// TIA Portal V18 export
FUNCTION_BLOCK "LEDS"   // FB17, LAD
{ S7_Optimized_Access := 'TRUE' }
// stored: AutoNumber false, MemoryReserve 100, SetENOAutomatically false
   VAR
      ElevClLEDStatus : Bool;
      MSVClLEDStatus : Bool;
      BUWClLEDStatus : Bool;
   END_VAR
   VAR_TEMP
      BUWClLEDOffDely : Bool;
   END_VAR
BEGIN

REGION Network 1: Elev Closed LED
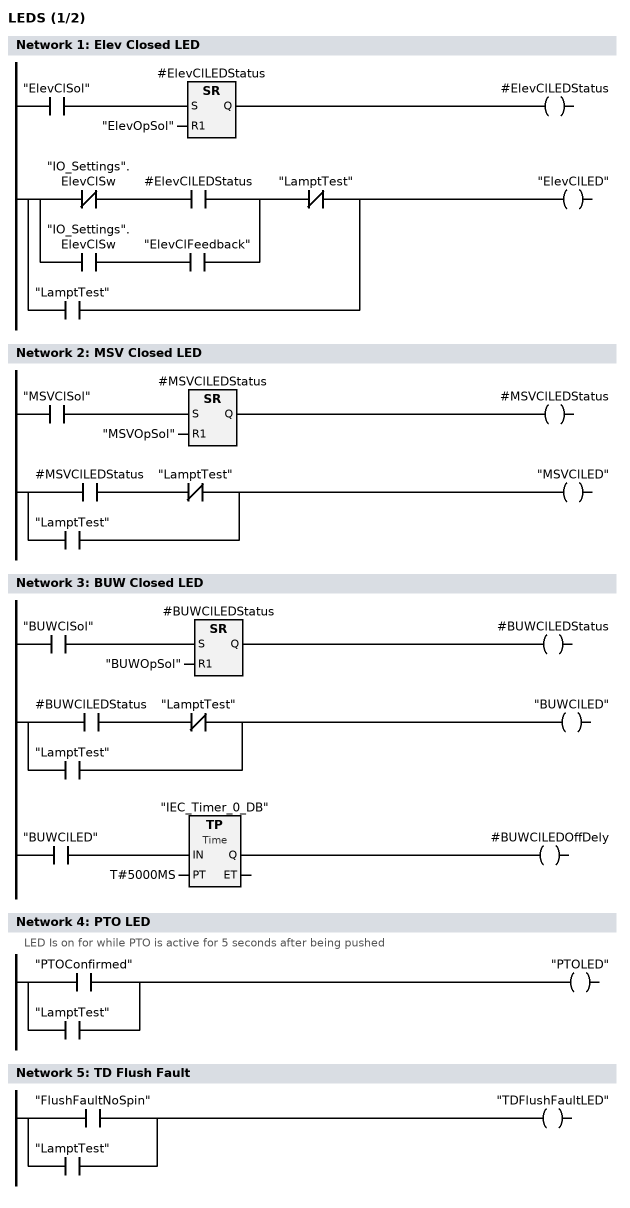
   RUNG wire#powerrail
      Contact( "ElevClSol" )
      S_SR(operand := #ElevClLEDStatus, r1 := "ElevOpSol")
      Coil( #ElevClLEDStatus )
   END_RUNG
   RUNG wire#powerrail
      I_Contact( "IO_Settings".ElevClSw )
      Contact( #ElevClLEDStatus )
      wire#w1
      I_Contact( "LamptTest" )
      wire#w2
      Coil( "ElevClLED" )
   END_RUNG
   RUNG wire#powerrail
      Contact( "IO_Settings".ElevClSw )
      Contact( "ElevClFeedback" )
   END_RUNG wire#w1
   RUNG wire#powerrail
      Contact( "LamptTest" )
   END_RUNG wire#w2
   // the same network as SCL:
   IF "ElevClSol" THEN
       #ElevClLEDStatus := TRUE;   // SR flip-flop
   END_IF;
   IF "ElevOpSol" THEN #ElevClLEDStatus := FALSE; END_IF;
   #ElevClLEDStatus := #ElevClLEDStatus;
   "ElevClLED" := (((NOT "IO_Settings".ElevClSw AND #ElevClLEDStatus) OR ("IO_Settings".ElevClSw AND "ElevClFeedback")) AND NOT "LamptTest") OR "LamptTest";
END_REGION

REGION Network 2: MSV Closed LED
   RUNG wire#powerrail
      Contact( "MSVClSol" )
      S_SR(operand := #MSVClLEDStatus, r1 := "MSVOpSol")
      Coil( #MSVClLEDStatus )
   END_RUNG
   RUNG wire#powerrail
      Contact( #MSVClLEDStatus )
      I_Contact( "LamptTest" )
      wire#w1
      Coil( "MSVClLED" )
   END_RUNG
   RUNG wire#powerrail
      Contact( "LamptTest" )
   END_RUNG wire#w1
   // the same network as SCL:
   IF "MSVClSol" THEN
       #MSVClLEDStatus := TRUE;   // SR flip-flop
   END_IF;
   IF "MSVOpSol" THEN #MSVClLEDStatus := FALSE; END_IF;
   #MSVClLEDStatus := #MSVClLEDStatus;
   "MSVClLED" := (#MSVClLEDStatus AND NOT "LamptTest") OR "LamptTest";
END_REGION

REGION Network 3: BUW Closed LED
   RUNG wire#powerrail
      Contact( "BUWClSol" )
      S_SR(operand := #BUWClLEDStatus, r1 := "BUWOpSol")
      Coil( #BUWClLEDStatus )
   END_RUNG
   RUNG wire#powerrail
      Contact( #BUWClLEDStatus )
      I_Contact( "LamptTest" )
      wire#w1
      Coil( "BUWClLED" )
   END_RUNG
   RUNG wire#powerrail
      Contact( "LamptTest" )
   END_RUNG wire#w1
   RUNG wire#powerrail
      Contact( "BUWClLED" )
      { S7_Templates := "time_type := Time" } "IEC_Timer_0_DB".TP(pt := T#5000MS, et =>)
      Coil( #BUWClLEDOffDely )
   END_RUNG
   // the same network as SCL:
   IF "BUWClSol" THEN
       #BUWClLEDStatus := TRUE;   // SR flip-flop
   END_IF;
   IF "BUWOpSol" THEN #BUWClLEDStatus := FALSE; END_IF;
   #BUWClLEDStatus := #BUWClLEDStatus;
   "BUWClLED" := (#BUWClLEDStatus AND NOT "LamptTest") OR "LamptTest";
   "IEC_Timer_0_DB".TP(IN := "BUWClLED", PT := T#5000MS);
   #BUWClLEDOffDely := "IEC_Timer_0_DB".Q;
END_REGION

REGION Network 4: PTO LED
   // LED Is on for while PTO is active for 5 seconds after being pushed
   RUNG wire#powerrail
      Contact( "PTOConfirmed" )
      wire#w1
      Coil( "PTOLED" )
   END_RUNG
   RUNG wire#powerrail
      Contact( "LamptTest" )
   END_RUNG wire#w1
   // the same network as SCL:
   "PTOLED" := "PTOConfirmed" OR "LamptTest";
END_REGION

REGION Network 5: TD Flush Fault
   RUNG wire#powerrail
      Contact( "FlushFaultNoSpin" )
      wire#w1
      Coil( "TDFlushFaultLED" )
   END_RUNG
   RUNG wire#powerrail
      Contact( "LamptTest" )
   END_RUNG wire#w1
   // the same network as SCL:
   "TDFlushFaultLED" := "FlushFaultNoSpin" OR "LamptTest";
END_REGION

REGION Network 6: Quill Lock LED
   // IF Quill Lock, Lock Maintained and BUW is closed,(LED is ON) then Quill Lock
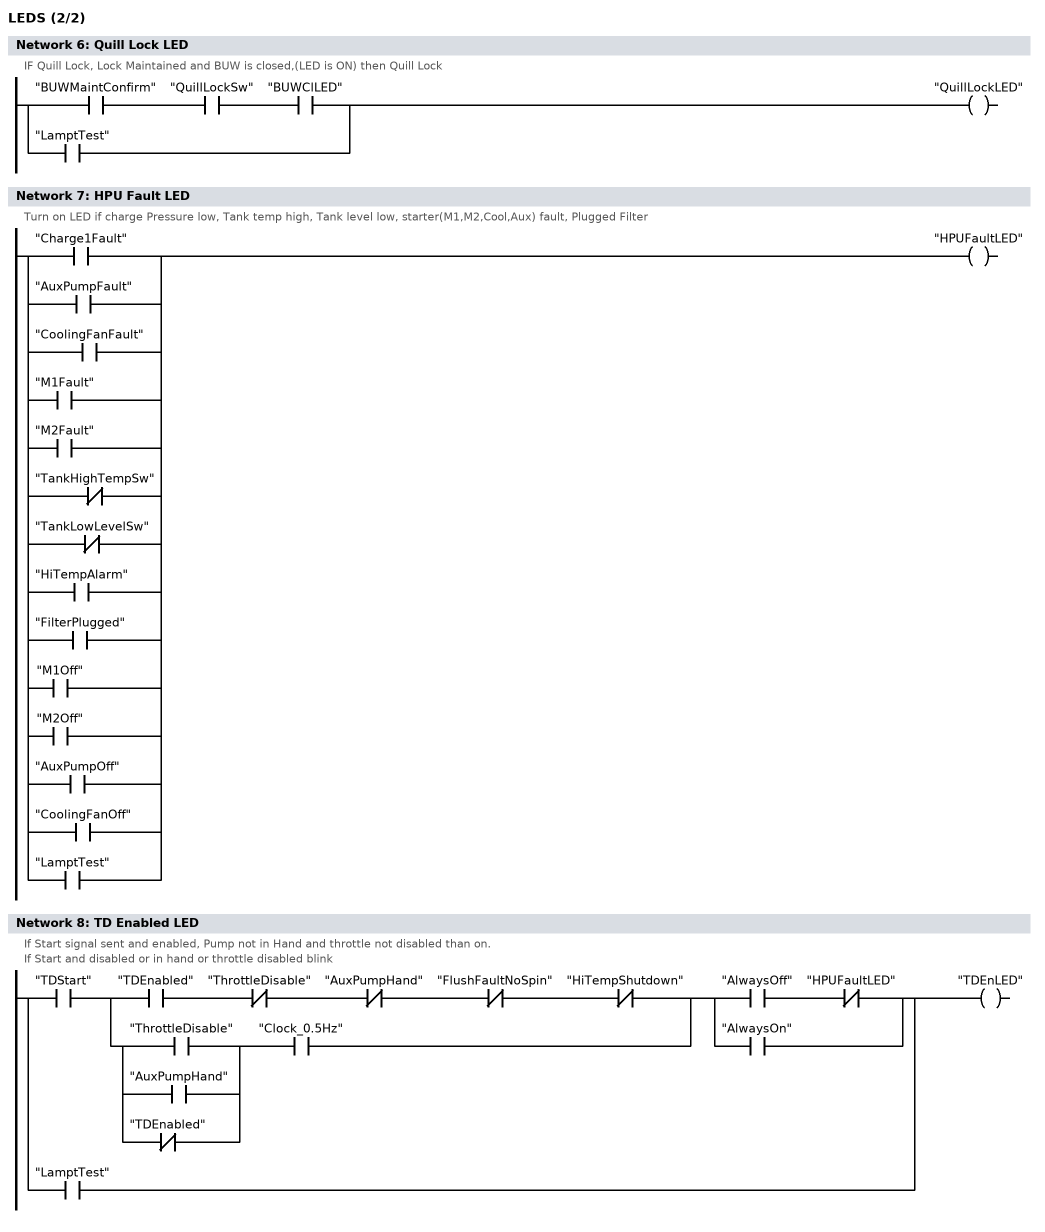
   RUNG wire#powerrail
      Contact( "BUWMaintConfirm" )
      Contact( "QuillLockSw" )
      Contact( "BUWClLED" )
      wire#w1
      Coil( "QuillLockLED" )
   END_RUNG
   RUNG wire#powerrail
      Contact( "LamptTest" )
   END_RUNG wire#w1
   // the same network as SCL:
   "QuillLockLED" := ("BUWMaintConfirm" AND "QuillLockSw" AND "BUWClLED") OR "LamptTest";
END_REGION

REGION Network 7: HPU Fault LED
   // Turn on LED if charge Pressure low, Tank temp high, Tank level low, starter(M1,M2,Cool,Aux) fault, Plugged Filter
   RUNG wire#powerrail
      Contact( "Charge1Fault" )
      wire#w1
      Coil( "HPUFaultLED" )
   END_RUNG
   RUNG wire#powerrail
      Contact( "AuxPumpFault" )
   END_RUNG wire#w1
   RUNG wire#powerrail
      Contact( "CoolingFanFault" )
   END_RUNG wire#w1
   RUNG wire#powerrail
      Contact( "M1Fault" )
   END_RUNG wire#w1
   RUNG wire#powerrail
      Contact( "M2Fault" )
   END_RUNG wire#w1
   RUNG wire#powerrail
      I_Contact( "TankHighTempSw" )
   END_RUNG wire#w1
   RUNG wire#powerrail
      I_Contact( "TankLowLevelSw" )
   END_RUNG wire#w1
   RUNG wire#powerrail
      Contact( "HiTempAlarm" )
   END_RUNG wire#w1
   RUNG wire#powerrail
      Contact( "FilterPlugged" )
   END_RUNG wire#w1
   RUNG wire#powerrail
      Contact( "M1Off" )
   END_RUNG wire#w1
   RUNG wire#powerrail
      Contact( "M2Off" )
   END_RUNG wire#w1
   RUNG wire#powerrail
      Contact( "AuxPumpOff" )
   END_RUNG wire#w1
   RUNG wire#powerrail
      Contact( "CoolingFanOff" )
   END_RUNG wire#w1
   RUNG wire#powerrail
      Contact( "LamptTest" )
   END_RUNG wire#w1
   // the same network as SCL:
   "HPUFaultLED" := "Charge1Fault" OR "AuxPumpFault" OR "CoolingFanFault" OR "M1Fault" OR "M2Fault" OR NOT "TankHighTempSw" OR NOT "TankLowLevelSw" OR "HiTempAlarm" OR "FilterPlugged" OR "M1Off" OR "M2Off" OR "AuxPumpOff" OR "CoolingFanOff" OR "LamptTest";
END_REGION

REGION Network 8: TD Enabled LED
   // If Start signal sent and enabled, Pump not in Hand and throttle not disabled than on. 
   // If Start and disabled or in hand or throttle disabled blink
   RUNG wire#powerrail
      Contact( "TDStart" )
      wire#w1
      Contact( "TDEnabled" )
      I_Contact( "ThrottleDisable" )
      I_Contact( "AuxPumpHand" )
      I_Contact( "FlushFaultNoSpin" )
      I_Contact( "HiTempShutdown" )
      wire#w2
      Contact( "AlwaysOff" )
      I_Contact( "HPUFaultLED" )
      wire#w4
      Coil( "TDEnLED" )
   END_RUNG
   RUNG wire#w1
      Contact( "ThrottleDisable" )
      wire#w3
      Contact( "Clock_0.5Hz" )
   END_RUNG wire#w2
   RUNG wire#w1
      Contact( "AuxPumpHand" )
   END_RUNG wire#w3
   RUNG wire#w1
      I_Contact( "TDEnabled" )
   END_RUNG wire#w3
   RUNG wire#w2
      Contact( "AlwaysOn" )
   END_RUNG wire#w4
   RUNG wire#powerrail
      Contact( "LamptTest" )
   END_RUNG wire#w4
   // the same network as SCL:
   "TDEnLED" := ("TDStart" AND (("TDEnabled" AND NOT "ThrottleDisable" AND NOT "AuxPumpHand" AND NOT "FlushFaultNoSpin" AND NOT "HiTempShutdown") OR (("ThrottleDisable" OR "AuxPumpHand" OR NOT "TDEnabled") AND "Clock_0.5Hz")) AND (("AlwaysOff" AND NOT "HPUFaultLED") OR "AlwaysOn")) OR "LamptTest";
END_REGION
END_FUNCTION_BLOCK
